(*
Interface for components that can be returned to a known initial state.

Implementors must define :meth:`Reset` to clear any internal state, such as
accumulators, filter history, or elapsed time, and restore the output to its
initial condition.
*)
INTERFACE I_Resettable EXTENDS __SYSTEM.IQueryInterface

(* Clears internal state and restores the component to its initial condition. *)
METHOD Reset
VAR_INPUT
END_VAR
END_METHOD

END_INTERFACE

(* stored: Version 1.1.0.1, ProductVersion 3.1.4024.15
   Itf I_Resettable: Id {ab5914ee-8b82-4d90-a04f-4fe8555aca42}
   Method Reset: Id {b7f6a5e4-6d73-4a58-a83e-a8644bfdc1ce} *)
